// TIA Portal V20 export
FUNCTION_BLOCK "Send_FData"   // FB3, FBD
{ S7_Optimized_Access := 'TRUE' }
// stored: MemoryReserve 100, SetENOAutomatically false
   VAR
      TSEND_Instance { S7_SetPoint := 'True'} : TSEND;
      status_save { S7_SetPoint := 'True'} : Word;
      trigger : Bool;
   END_VAR
   VAR_TEMP   // added for the SCL form of the ladder/FBD networks
      _w1 : Bool;
   END_VAR
BEGIN

REGION Network 1
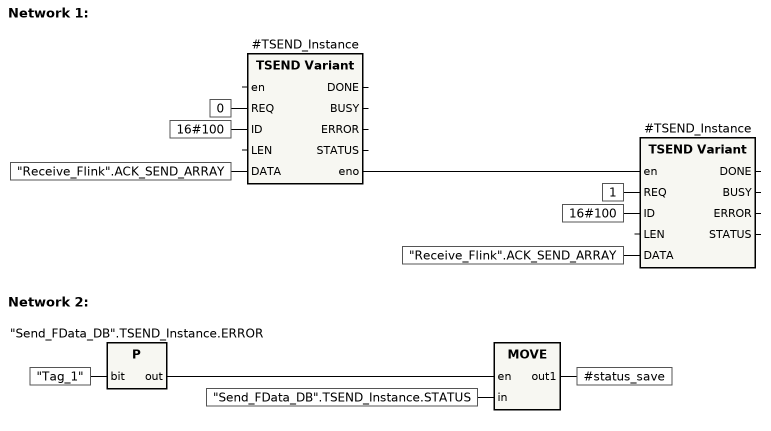
   #TSEND_Instance(REQ := 0, ID := 16#100, DATA := "Receive_Flink".ACK_SEND_ARRAY, ENO => #_w1);   // TSEND
   IF #_w1 THEN
       #TSEND_Instance(REQ := 1, ID := 16#100, DATA := "Receive_Flink".ACK_SEND_ARRAY);   // TSEND
   END_IF;
END_REGION

REGION Network 2
   #_w1 := "Send_FData_DB".TSEND_Instance.ERROR AND NOT "Tag_1";   // rising edge of "Send_FData_DB".TSEND_Instance.ERROR
   "Tag_1" := "Send_FData_DB".TSEND_Instance.ERROR;
   IF #_w1 THEN #status_save := "Send_FData_DB".TSEND_Instance.STATUS; END_IF;
END_REGION
END_FUNCTION_BLOCK
